KUKA KRL data list: ros_krlptp.dat

&ACCESS RVP
&REL 101
&PARAM DISKPATH = KRC:\R1\Program\ROS
DEFDAT  ROS_KRLPTP PUBLIC
INT movesQueued=0
REAL moveTime=0.0360000
REAL moveTime2=0.104000
E6AXIS nextMove={A1 -106.622528,A2 -31.4800682,A3 -40.7959671,A4 -36.6705093,A5 72.0757370,A6 139.748947,E1 -0.00564089,E2 0.00186683913,E3 0.0,E4 0.0,E5 0.0,E6 0.0}
DECL PDAT ROS_Pdat={VEL 50.0000,ACC 50.0000,APO_DIST 20.0000,GEAR_JERK 100.000,EXAX_IGN 0}
ENDDAT
